FUNCTION_BLOCK BasicWithAdapter
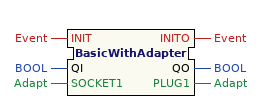
  EVENT_INPUT
    INIT;
  END_EVENT
  EVENT_OUTPUT
    INITO;
  END_EVENT
  VAR_INPUT
    QI : BOOL;
  END_VAR
  VAR_OUTPUT
    QO : BOOL;
  END_VAR
  SOCKETS
    SOCKET1 : Adapt;
  END_SOCKETS
  PLUGS
    PLUG1 : Adapt;
  END_PLUGS
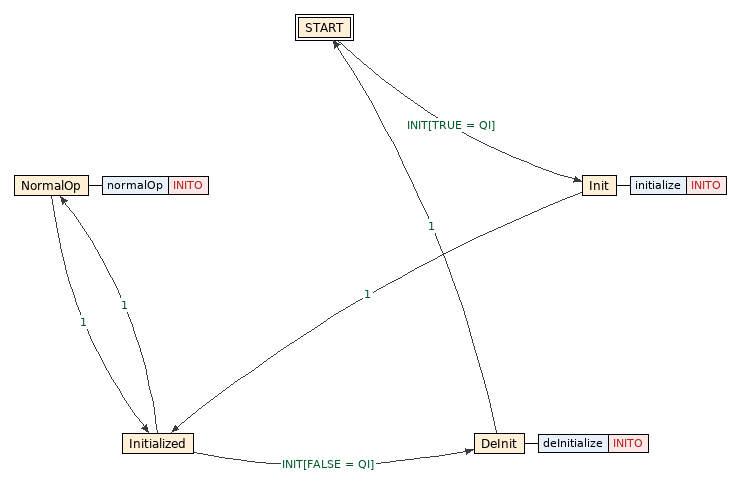
  EC_STATES
    START;
    Init : initialize -> INITO;
    DeInit : deInitialize -> INITO;
    Initialized;
    NormalOp : normalOp -> INITO;
  END_STATES
  EC_TRANSITIONS
    START TO Init := INIT[TRUE = QI];
    Init TO Initialized := 1;
    Initialized TO NormalOp := 1;
    NormalOp TO Initialized := 1;
    Initialized TO DeInit := INIT[FALSE = QI];
    DeInit TO START := 1;
  END_TRANSITIONS
  ALGORITHM initialize IN ST:
QO := QI;&#38;#10;
  END_ALGORITHM
  ALGORITHM normalOp IN ST:
QO := QI;&#38;#10;
  END_ALGORITHM
  ALGORITHM deInitialize IN ST:
QO := FALSE;&#38;#10;
  END_ALGORITHM
END_FUNCTION_BLOCK
